FUNCTION_BLOCK UDP_LISTEN (* Listener for a Multicast UDP Socket *)
  (* Standard: 61499-1; Classification: Communications; ApplicationDomain: Feasibility Demo *)
  (* Version 0.2, 2001-05-25, JHC, Rockwell Automation, Added service sequences. *)
  (* Version 0.1, 2000-05-16, JHC, Rockwell Automation, File type changed to ".fbt" *)
  (* Version 0.0, 2000-03-30, JHC, Rockwell Automation *)
  (* Compiler header: package fb.rt.ita; import java.io.*; import fb.rt.net.*; *)
  (* Compiler classdef: public class UDP_LISTEN extends SUBSCRIBE_0 implements Runnable *)
  (* Compiler Java IBM VisualAge 3.0 *)
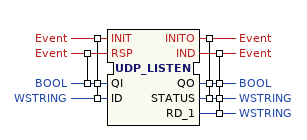
  EVENT_INPUT
    INIT WITH QI, ID; (* Service Initialization *)
    RSP WITH QI; (* Service Response *)
  END_EVENT
  EVENT_OUTPUT
    INITO WITH QO, STATUS; (* Initialization Confirm *)
    IND WITH QO, STATUS, RD_1; (* Message received *)
  END_EVENT
  VAR_INPUT
    QI : BOOL; (* Event Input Qualifier *)
    ID : WSTRING; (* Connection Identifier *)
  END_VAR
  VAR_OUTPUT
    QO : BOOL; (* Event Output Qualifier *)
    STATUS : WSTRING; (* Service Status *)
    RD_1 : WSTRING; (* Message in Hex up to trailing zeroes *)
  END_VAR
  SERVICE PUBLISH_x/UDP_LISTEN (* Data Monitoring Service *)
    SEQUENCE normal_establishment
      PUBLISH_x.INIT+(ID) -> PUBLISH_x.INITO+();
      UDP_LISTEN.INIT+(ID) -> UDP_LISTEN.INITO+();
    END_SEQUENCE
    SEQUENCE publisher_rejected_establishment
      PUBLISH_x.INIT+(ID) -> PUBLISH_x.INITO-(STATUS);
    END_SEQUENCE
    SEQUENCE subscriber_rejected_establishment
      UDP_LISTEN.INIT+(ID) -> UDP_LISTEN.INITO-(STATUS);
    END_SEQUENCE
    SEQUENCE normal_data_transfer
      PUBLISH_x.REQ+(SD_1) -> UDP_LISTEN.IND+(RD_1);
      -> PUBLISH_x.CNF+();
      UDP_LISTEN.RSP+();
    END_SEQUENCE
    SEQUENCE data_transfer_error
      PUBLISH_x.REQ+(SD_1) -> UDP_LISTEN.IND-(STATUS);
      -> PUBLISH_x.CNF+();
    END_SEQUENCE
    SEQUENCE publisher_initiated_disconnect
      PUBLISH_x.INIT-() -> UDP_LISTEN.INITO-(STATUS);
      -> PUBLISH_x.INITO-(STATUS);
    END_SEQUENCE
    SEQUENCE subscriber_initiated_disconnect
      UDP_LISTEN.INIT-() -> UDP_LISTEN.INITO-(STATUS);
    END_SEQUENCE
    SEQUENCE system_publisher_disconnect
      -> PUBLISH_x.INITO-(STATUS);
      -> UDP_LISTEN.INITO-(STATUS);
    END_SEQUENCE
    SEQUENCE system_subscriber_disconnect
      -> UDP_LISTEN.INITO-(STATUS);
    END_SEQUENCE
  END_SERVICE
END_FUNCTION_BLOCK
